INTERFACE I_CameraTriggerDevice

METHOD CamTrigger
VAR_INPUT
  bOk             : BOOL;     // trigger is ok
	nPos            : DINT;     // camera triggered position
  nPosDeviation   : DINT;     // camera started deviation
END_VAR
END_METHOD

METHOD CamTriggerDone
VAR_INPUT
END_VAR
END_METHOD

{attribute 'monitoring':='call'}
PROPERTY fTriggerDistance : LREAL
GET
END_GET
END_PROPERTY

PROPERTY fTriggerPulseLength : LREAL
GET
END_GET
END_PROPERTY

END_INTERFACE

(* stored: Version 1.1.0.1, ProductVersion 3.1.4024.3
   Itf I_CameraTriggerDevice: Id {9a227b26-fb89-41d0-9430-738990902071}
   Method CamTrigger: Id {1ddb9edf-d457-4eaf-bfb5-deaddecb3a6e}
   Method CamTriggerDone: Id {5a50f2bd-1e69-4810-a974-cfd3eb90e67c}
   Property fTriggerDistance: Id {b1019d44-af6e-4e69-afdc-ed26fe213b6a}
   Get Get: Id {bedcfbe6-faaf-4600-b433-0455bcc90f7f}
   Property fTriggerPulseLength: Id {e18b5776-7f0a-4909-bcb4-39a3beb5b879}
   Get Get: Id {67c85c5c-3706-4e0a-85f8-7b21a3e7ab83} *)
